Staubli VAL3: refresh.pgx

program refresh()
// // page refresh
begin
  if !use:bShowDialog and !cycleStatus:bShowMessage
    //
    // refresh the static message
    if (nKey>=270 and nKey<=278)or(use:bUseRefresh and !bShowStatus)or(nKey>=261 and nKey<=269)
      call buildList()
      call refreshStatic()
      call refreshDynamic()
    else
      if !bShowStatus
        // refresh the Dynamic message
        if abs(clock()-nRefresh)>nTime
          call refreshDynamic()
        endIf
      endIf
    endIf
    //
    call showStatus()
  endIf
end
